// TIA Portal V17 export
// export: Created 2022-02-03T14:45:12.5581156Z, ExportSetting WithDefaults, DisplayName Totally Integrated Automation Portal, DisplayVersion V17, DisplayName TIA Portal Openness, DisplayVersion V17, DisplayName TIA Portal Version Control Interface, DisplayVersion V17, DisplayName SINAMICS Startdrive Advanced, DisplayVersion V17, DisplayName SINAMICS Startdrive G130, G150, S120, S150, SINAMICS MV, S210, DisplayVersion V17, DisplayName SINAMICS Startdrive G110M, G120, G120C, G120D, G120P, G115D, DisplayVersion V17, DisplayName STEP 7 Professional, DisplayVersion V17, DisplayName STEP 7 Safety, DisplayVersion V17, DisplayName WinCC Advanced, DisplayVersion V17
ORGANIZATION_BLOCK "MainWeight"   // OB125, LAD, ProgramCycle
TITLE = "Main Program Sweep (Cycle)"
VERSION : 0.1
// stored: AutoNumber true, IsIECCheckEnabled false, SetENOAutomatically false
   VAR_INPUT
      Initial_Call : Bool;   // Initial call of this OB
      Remanence : Bool;   // =True, if remanent data are available
   END_VAR
BEGIN

REGION Network 1
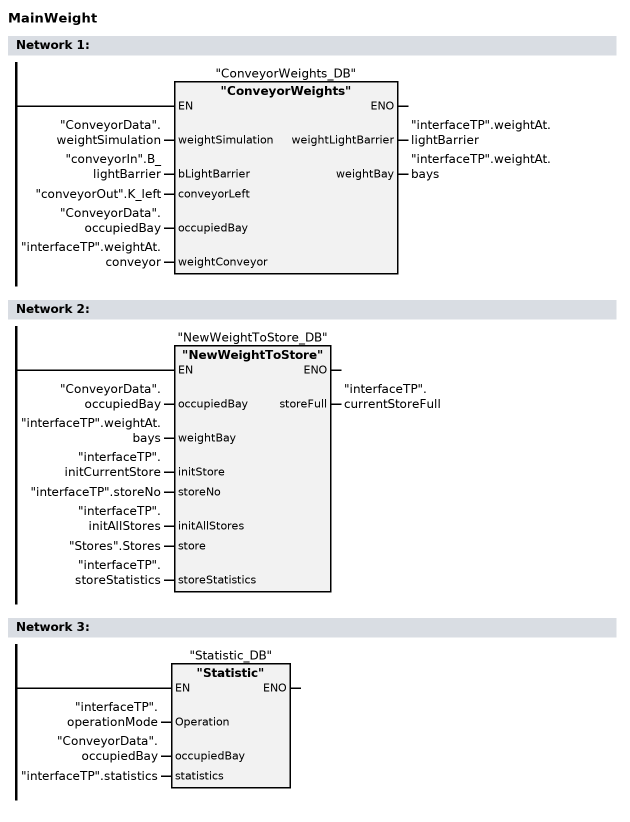
   RUNG wire#powerrail
      "ConveyorWeights_DB"(weightSimulation := "ConveyorData".weightSimulation, bLightBarrier := "conveyorIn".B_lightBarrier, conveyorLeft := "conveyorOut".K_left, occupiedBay := "ConveyorData".occupiedBay, weightConveyor := "interfaceTP".weightAt.conveyor, weightLightBarrier => "interfaceTP".weightAt.lightBarrier, weightBay => "interfaceTP".weightAt.bays)
   END_RUNG
   // the same network as SCL:
   "ConveyorWeights_DB"(weightSimulation := "ConveyorData".weightSimulation,   // "ConveyorWeights"
                        bLightBarrier := "conveyorIn".B_lightBarrier,
                        conveyorLeft := "conveyorOut".K_left,
                        occupiedBay := "ConveyorData".occupiedBay,
                        weightConveyor := "interfaceTP".weightAt.conveyor,
                        weightLightBarrier => "interfaceTP".weightAt.lightBarrier,
                        weightBay => "interfaceTP".weightAt.bays);
END_REGION

REGION Network 2
   RUNG wire#powerrail
      "NewWeightToStore_DB"(occupiedBay := "ConveyorData".occupiedBay, weightBay := "interfaceTP".weightAt.bays, initStore := "interfaceTP".initCurrentStore, storeNo := "interfaceTP".storeNo, initAllStores := "interfaceTP".initAllStores, store := "Stores".Stores, storeStatistics := "interfaceTP".storeStatistics, storeFull => "interfaceTP".currentStoreFull)
   END_RUNG
   // the same network as SCL:
   "NewWeightToStore_DB"(occupiedBay := "ConveyorData".occupiedBay,   // "NewWeightToStore"
                         weightBay := "interfaceTP".weightAt.bays,
                         initStore := "interfaceTP".initCurrentStore,
                         storeNo := "interfaceTP".storeNo,
                         initAllStores := "interfaceTP".initAllStores,
                         store := "Stores".Stores,
                         storeStatistics := "interfaceTP".storeStatistics,
                         storeFull => "interfaceTP".currentStoreFull);
END_REGION

REGION Network 3
   RUNG wire#powerrail
      "Statistic_DB"(Operation := "interfaceTP".operationMode, occupiedBay := "ConveyorData".occupiedBay, statistics := "interfaceTP".statistics)
   END_RUNG
   // the same network as SCL:
   "Statistic_DB"(Operation := "interfaceTP".operationMode,   // "Statistic"
                  occupiedBay := "ConveyorData".occupiedBay,
                  statistics := "interfaceTP".statistics);
END_REGION
END_ORGANIZATION_BLOCK
